// TIA Portal project "noe_red" (V15)

(* hardware
DEVICE "S7-1200 station_1"  S7-1200 Station
   slot 0: "Rack_0"  S7-1200 Rack  Rack  V1.0
   slot 1: "PLC_1"  CPU 1214C DC/DC/DC  6ES7 214-1AG40-0XB0  V4.2
*)

// ===== PLC "PLC_1"  CPU 1214C DC/DC/DC =====

VAR_GLOBAL   // PLC tag table "int/out_plc"
   "Led1" AT %Q0.0 : Bool;
   "Led2" AT %Q0.1 : Bool;
   "Led3" AT %Q0.2 : Bool;
   "Led4" AT %Q0.3 : Bool;
   "Led5" AT %Q0.4 : Bool;
   "Led6" AT %Q0.5 : Bool;
   "Led7" AT %Q0.6 : Bool;
   "Led8" AT %Q0.7 : Bool;
   "Led9" AT %Q1.0 : Bool;
   "Led10" AT %Q1.1 : Bool;
   "sensor_1" AT %I0.0 : Bool;
   "sensor_2" AT %I0.1 : Bool;
   "sensor_3" AT %I0.2 : Bool;
   "sensor_4" AT %I0.3 : Bool;
   "sensor_5" AT %I0.4 : Bool;
   "sensor_6" AT %I0.5 : Bool;
   "sensor_7" AT %I0.6 : Bool;
   "sensor_8" AT %I0.7 : Bool;
   "sensor_9" AT %I1.0 : Bool;
   "sensor_10" AT %I1.1 : Bool;
   "sensor_11" AT %I1.2 : Bool;
   "sensor_12" AT %I1.3 : Bool;
   "sensor_13" AT %I1.4 : Bool;
   "sensor_14" AT %I1.5 : Bool;
   "System_Byte" AT %MB1000 : Byte;
   "FirstScan" AT %M1000.0 : Bool;
   "DiagStatusUpdate" AT %M1000.1 : Bool;
   "AlwaysTRUE" AT %M1000.2 : Bool;
   "AlwaysFALSE" AT %M1000.3 : Bool;
   "Clock_Byte" AT %MB1001 : Byte;
   "Clock_10Hz" AT %M1001.0 : Bool;
   "Clock_5Hz" AT %M1001.1 : Bool;
   "Clock_2.5Hz" AT %M1001.2 : Bool;
   "Clock_2Hz" AT %M1001.3 : Bool;
   "Clock_1.25Hz" AT %M1001.4 : Bool;
   "Clock_1Hz" AT %M1001.5 : Bool;
   "Clock_0.625Hz" AT %M1001.6 : Bool;
   "Clock_0.5Hz" AT %M1001.7 : Bool;
END_VAR

VAR_GLOBAL   // PLC tag table "varible_m_control_plc"
   "var_out_0" AT %M1.0 : Bool;
   "var_out_1" AT %M1.1 : Bool;
   "var_out_2" AT %M1.2 : Bool;
   "var_out_3" AT %M1.3 : Bool;
   "var_out_4" AT %M1.4 : Bool;
   "var_out_5" AT %M1.5 : Bool;
   "var_out_6" AT %M1.6 : Bool;
   "var_out_7" AT %M1.7 : Bool;
   "var_out_8" AT %M2.0 : Bool;
   "var_out_9" AT %M2.1 : Bool;
   "var_out_10" AT %M2.2 : Bool;
   "var_in_0" AT %M3.0 : Bool;
   "var_in_1" AT %M3.1 : Bool;
   "var_in_2" AT %M3.2 : Bool;
   "var_in_3" AT %M3.3 : Bool;
   "var_in_4" AT %M3.4 : Bool;
   "var_in_5" AT %M3.5 : Bool;
   "var_in_6" AT %M3.6 : Bool;
   "var_in_7" AT %M3.7 : Bool;
   "var_in_8" AT %M4.0 : Bool;
   "var_in_9" AT %M4.1 : Bool;
   "var_in_10" AT %M4.2 : Bool;
   "var_in_11" AT %M4.3 : Bool;
   "var_in_12" AT %M4.4 : Bool;
   "var_in_13" AT %M4.5 : Bool;
   "var_in_14" AT %M4.6 : Bool;
END_VAR

ORGANIZATION_BLOCK "Main"   // OB1, LAD, ProgramCycle
TITLE = "Main Program Sweep (Cycle)"
{ S7_Optimized_Access := 'TRUE' }
VERSION : 0.1
   VAR_INPUT
      Initial_Call : Bool;   // Initial call of this OB
      Remanence : Bool;   // =True, if remanent data are available
   END_VAR
BEGIN

REGION Network 1
   // control in/output plc  by Node_Red
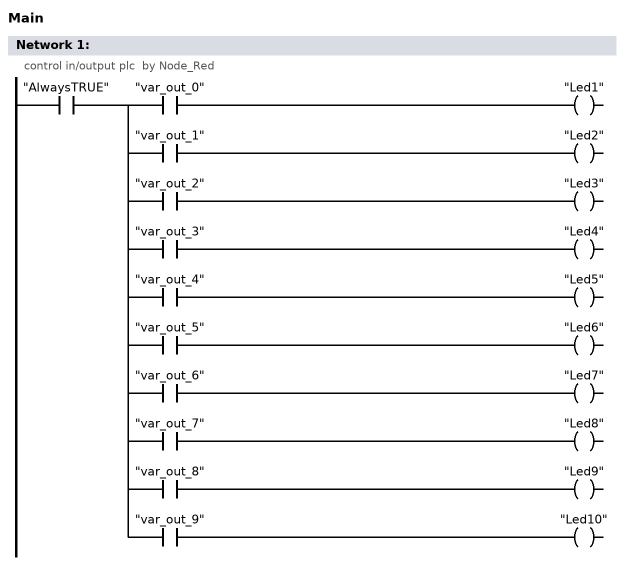
   RUNG wire#powerrail
      Contact( "AlwaysTRUE" )
      wire#w1
      Contact( "var_out_0" )
      Coil( "Led1" )
   END_RUNG
   RUNG wire#w1
      Contact( "var_out_1" )
      Coil( "Led2" )
   END_RUNG
   RUNG wire#w1
      Contact( "var_out_2" )
      Coil( "Led3" )
   END_RUNG
   RUNG wire#w1
      Contact( "var_out_3" )
      Coil( "Led4" )
   END_RUNG
   RUNG wire#w1
      Contact( "var_out_4" )
      Coil( "Led5" )
   END_RUNG
   RUNG wire#w1
      Contact( "var_out_5" )
      Coil( "Led6" )
   END_RUNG
   RUNG wire#w1
      Contact( "var_out_6" )
      Coil( "Led7" )
   END_RUNG
   RUNG wire#w1
      Contact( "var_out_7" )
      Coil( "Led8" )
   END_RUNG
   RUNG wire#w1
      Contact( "var_out_8" )
      Coil( "Led9" )
   END_RUNG
   RUNG wire#w1
      Contact( "var_out_9" )
      Coil( "Led10" )
   END_RUNG
   // the same network as SCL:
   "Led1" := "AlwaysTRUE" AND "var_out_0";
   "Led2" := "AlwaysTRUE" AND "var_out_1";
   "Led3" := "AlwaysTRUE" AND "var_out_2";
   "Led4" := "AlwaysTRUE" AND "var_out_3";
   "Led5" := "AlwaysTRUE" AND "var_out_4";
   "Led6" := "AlwaysTRUE" AND "var_out_5";
   "Led7" := "AlwaysTRUE" AND "var_out_6";
   "Led8" := "AlwaysTRUE" AND "var_out_7";
   "Led9" := "AlwaysTRUE" AND "var_out_8";
   "Led10" := "AlwaysTRUE" AND "var_out_9";
END_REGION
END_ORGANIZATION_BLOCK